FUNCTION ReplaceAllAny
VAR_INPUT
	in : ANY;
	replaced : T_MaxString;
	with : T_MaxString;
END_VAR

ReplaceAllAnyType(in, replaced, with);

END_FUNCTION

(* stored: Version 1.1.0.1
   POU ReplaceAllAny: Id {4dfe1242-7df8-0cc0-1e8f-c32f9f237b90}, SpecialFunc None *)
